{attribute 'qualified_only'}
{attribute 'strict'}
{attribute 'to_string'}
TYPE E_FaultSeverity :
(
	CRITICAL,
	MINOR,
	MAJOR,
    WARNING
);
END_TYPE

(* stored: Version 1.1.0.1, ProductVersion 3.1.4026.18
   DUT E_FaultSeverity: Id {9c6627f8-acd0-45ba-849a-4769941fad65} *)
